SUBAPPLICATION AX_TO_QXA_BG_PUBLISH_SWITCHPIC (* AX_TO_QXA_BG_PUBLISH (Ausgang+Hintergrund+Publish) UND AX_SwitchPic_2_1 (ObjectPointer-Statusanzeige) aus demselben fertigen AX-Zustand gespeist - AX_SPLIT_2 davor, da beide Sub-Bausteine den Zustand brauchen (Adapter-Fanout-Regel). *)
  (* Standard: 61499-2; Description: Copyright (c) 2026 Meisterschulen am Ostbahnhof This program and the accompanying materials are made available under the terms of the Eclipse Public License 2.0 which is available at https://www.eclipse.org/legal/epl-2.0/ SPDX-License-Identifier: EPL-2.0 *)
  (* Version 1.0, 2026-09-17, Franz Höpfinger, Meisterschulen am Ostbahnhof, Neu (Franz: 'AX_TO_QXA_BG_PUBLISH AX_SPLIT_2 AX_SwitchPic_2_1 immer je in eine Subapp. wird eh 3x die gleiche') - aus Baender_EinAus.SUB herausgeloest, dort 3x identisch (Igel/Elevator/Querband) vorhanden. *)
  PACKAGE MyLib::sys;
  IMPORT isobus::UT::Q::const::IDs::ID_NULL;
  IMPORT logiBUS::io::DQ::logiBUS_DO;
  IMPORT logiBUS::io::DQ::logiBUS_DO_S;
  IMPORT isobus::UT::Q::types::s2x1ObjectIDs;
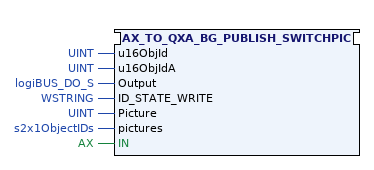
  VAR_INPUT
    u16ObjId : UINT := ID_NULL; (* Object ID Softkey - traegt die Hintergrundfarbe *)
    u16ObjIdA : UINT := ID_NULL; (* Object ID AuxFunction2 (Joystick) - zeigt Hintergrundfarbe am Aux-Handle mit *)
    Output : logiBUS::io::DQ::logiBUS_DO_S := logiBUS_DO::Invalid; (* Identify the Output Output_Q1..Q12 *)
    ID_STATE_WRITE : WSTRING; (* Lokale Publish-Adresse (ACTION=WRITE) fuer den tatsaechlichen Zustand - wird von Web-Client/Dashboard remote abonniert *)
    Picture : UINT; (* Object ID des ObjectPointer, der den Status-Kaestchen-Inhalt traegt *)
    pictures : isobus::UT::Q::types::s2x1ObjectIDs := (up := (u16ObjId := ID_NULL), down := (u16ObjId := ID_NULL)); (* die beiden Ziel-Object-IDs (up=aus, down=an) *)
  END_VAR
  SOCKETS
    IN : adapter::types::unidirectional::AX; (* Fertiger AX-Zustand (bereits zusammengefuehrt) - wird auf Ausgang+Hintergrund+Publish UND ObjectPointer-Statusanzeige verteilt *)
  END_SOCKETS
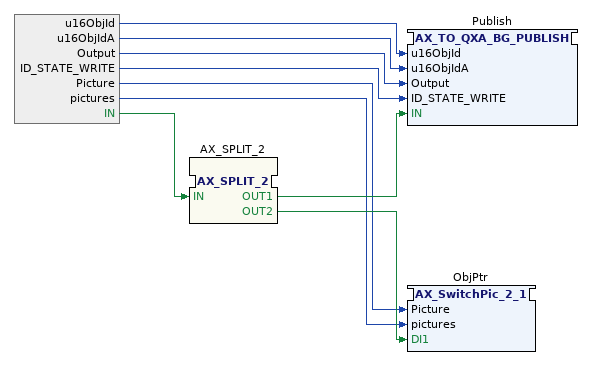
  FBS
    AX_SPLIT_2 : adapter::events::unidirectional::AX_SPLIT_2;
  END_FBS
  SUBAPPS
    Publish : MyLib::sys::AX_TO_QXA_BG_PUBLISH;
    ObjPtr : MyLib::sys::AX_SwitchPic_2_1;
  END_SUBAPPS
  DATA_CONNECTIONS
    u16ObjId TO Publish.u16ObjId;
    u16ObjIdA TO Publish.u16ObjIdA;
    Output TO Publish.Output;
    ID_STATE_WRITE TO Publish.ID_STATE_WRITE;
    Picture TO ObjPtr.Picture;
    pictures TO ObjPtr.pictures;
  END_CONNECTIONS
  ADAPTER_CONNECTIONS
    IN TO AX_SPLIT_2.IN;
    AX_SPLIT_2.OUT1 TO Publish.IN;
    AX_SPLIT_2.OUT2 TO ObjPtr.DI1;
  END_CONNECTIONS
END_SUBAPPLICATION
